FUNCTION_BLOCK ADD_3514EB543E3A8D7A (* Add *)
  (* Standard: 61499-2 *)
  (* Version 1.1, 24.06.2019, winkhub, nxtControl GmbH, support TIME *)
  PACKAGE Main;
  (* Compiler Cpp *)
  {SET_ATTRIBUTE(Runtime.FBType.ImplementingType, Runtime.Standard#DYNGEN_ADD)}
  {SET_ATTRIBUTE(Configuration.GenericFBType.InterfaceParams, Runtime.Standard#CNT:=5;IN${CNT$}:INT)}
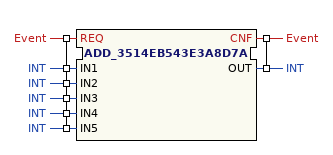
  EVENT_INPUT
    REQ WITH IN1, IN2, IN3, IN4, IN5; (* Normal Execution Request *)
  END_EVENT
  EVENT_OUTPUT
    CNF WITH OUT; (* Execution Confirmation *)
  END_EVENT
  VAR_INPUT
    IN1 : INT; (* Argument *)
    IN2 : INT; (* Argument *)
    IN3 : INT; (* Argument *)
    IN4 : INT; (* Argument *)
    IN5 : INT; (* Argument *)
  END_VAR
  VAR_OUTPUT
    OUT : INT; (* Result: IN1 + IN2 + ... *)
  END_VAR
  EC_STATES
    START;
  END_STATES
END_FUNCTION_BLOCK
